{attribute 'GeneratedUsingTerminal: EPP4314-1002-0016'}
{attribute addProperty BoxType "EPP4314-1002-0016"}
{attribute addProperty Id "InputAT %I*ARRAY[0..1] OF BOOL2TxPDO_StateAT %I*BOOL1TxPDO_ToggleAT %I*BOOL1"}
{attribute addProperty CRC "2573189997"}
{attribute addProperty Size "4"}
TYPE DI_Inputs_1F3A9325 :
STRUCT
	{attribute addProperty Name "Input"}
	Input AT %I* : ARRAY[0..1] OF BOOL;
	{attribute addProperty Name "TxPDO_State"}
	TxPDO_State AT %I* : BOOL;
	{attribute addProperty Name "TxPDO_Toggle"}
	TxPDO_Toggle AT %I* : BOOL;
END_STRUCT
END_TYPE

(* stored: Version 1.2.0.0, ProductVersion 3.1.4024.9
   DUT DI_Inputs_1F3A9325: Id {73b33d0d-aa82-4147-bad9-a4db31411a2b} *)
